(* Logix 5000 project; controller Amvex_Thorpe_Flowmeter vendor 1 type 14 code 106 rev 33.13; software revision 33.01; part 7 of 16 *)

ADD_ON_INSTRUCTION SetCheckpoint   (* revision 0.1, vendor Mecademic Inc., ExecuteEnableInFalse *)
// Inserts a "set checkpoint" command between two moves, so robot status reports that checkpoint id when reaching that command in the queue
VAR_IN_OUT
   RobotInputs : _061D:Meca500_86BDA20B:I:0; {required}
   RobotOutputs : _061D:Meca500_01F88326:O:0; {required}
END_VAR
VAR_INPUT
   Parameter_Value : REAL; {required}
   ExternalStateControl : BOOL; {required}
   ExternalMoveID : INT; {required}
END_VAR
VAR_OUTPUT
   Enabled : BOOL; {visible}
   Sent : BOOL; {visible}
   Buffered : BOOL; {visible}
   Error : BOOL; {visible}
END_VAR
VAR
   InternalMoveID : INT; {access None}
   MoveIDTrig : BOOL; {access None}
   MoveIDUpdated : BOOL; {access None}
   OneShot : DINT; {access None}
   FirstScan : BOOL; {access None}
END_VAR

ROUTINE EnableInFalse   (* ladder *)
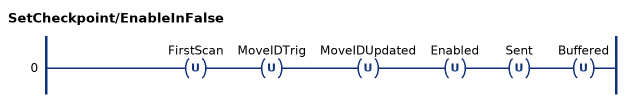
   0: OTU(FirstScan)OTU(MoveIDTrig)OTU(MoveIDUpdated)OTU(Enabled)OTU(Sent)OTU(Buffered);
END_ROUTINE

ROUTINE Logic   (* ladder *)
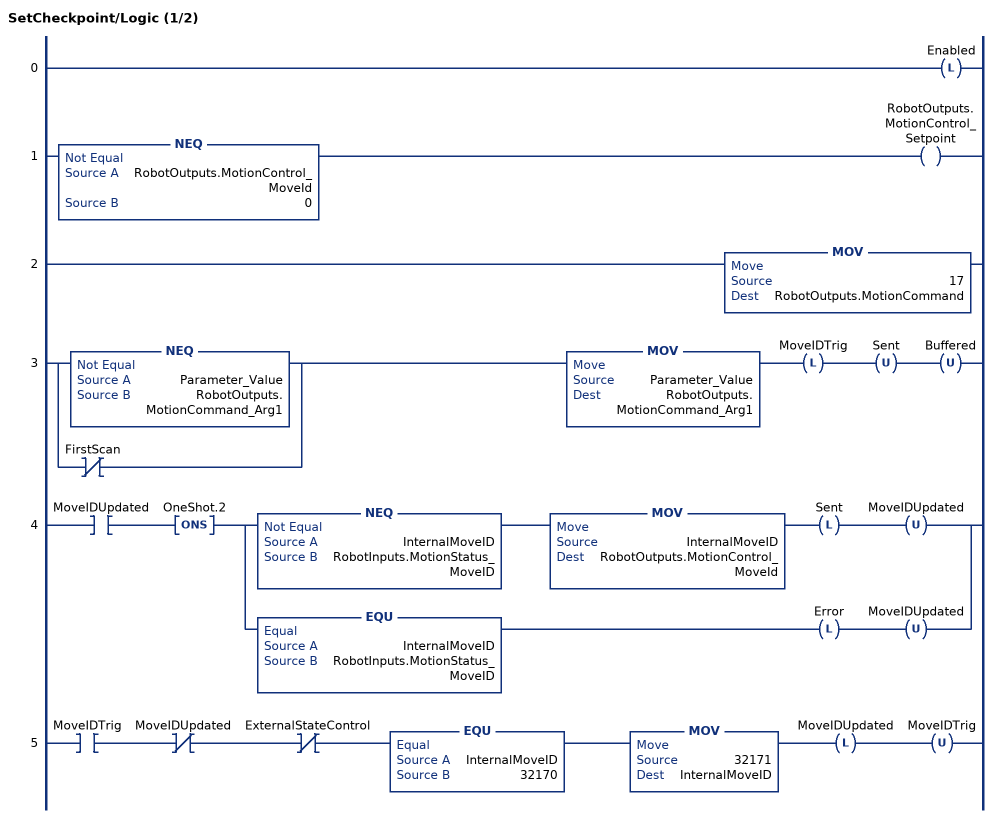
   0: OTL(Enabled);
   1: NEQ(RobotOutputs.MotionControl_MoveId,0)OTE(RobotOutputs.MotionControl_Setpoint);
   2: MOV(17,RobotOutputs.MotionCommand);
   3: [NEQ(Parameter_Value,RobotOutputs.MotionCommand_Arg1) ,XIO(FirstScan) ]MOV(Parameter_Value,RobotOutputs.MotionCommand_Arg1)OTL(MoveIDTrig)OTU(Sent)OTU(Buffered);
   4: XIC(MoveIDUpdated)ONS(OneShot.2)[NEQ(InternalMoveID,RobotInputs.MotionStatus_MoveID) MOV(InternalMoveID,RobotOutputs.MotionControl_MoveId) OTL(Sent) OTU(MoveIDUpdated) ,EQU(InternalMoveID,RobotInputs.MotionStatus_MoveID) OTL(Error) OTU(MoveIDUpdated) ];
   5: XIC(MoveIDTrig)XIO(MoveIDUpdated)XIO(ExternalStateControl)EQU(InternalMoveID,32170)MOV(32171,InternalMoveID)OTL(MoveIDUpdated)OTU(MoveIDTrig);
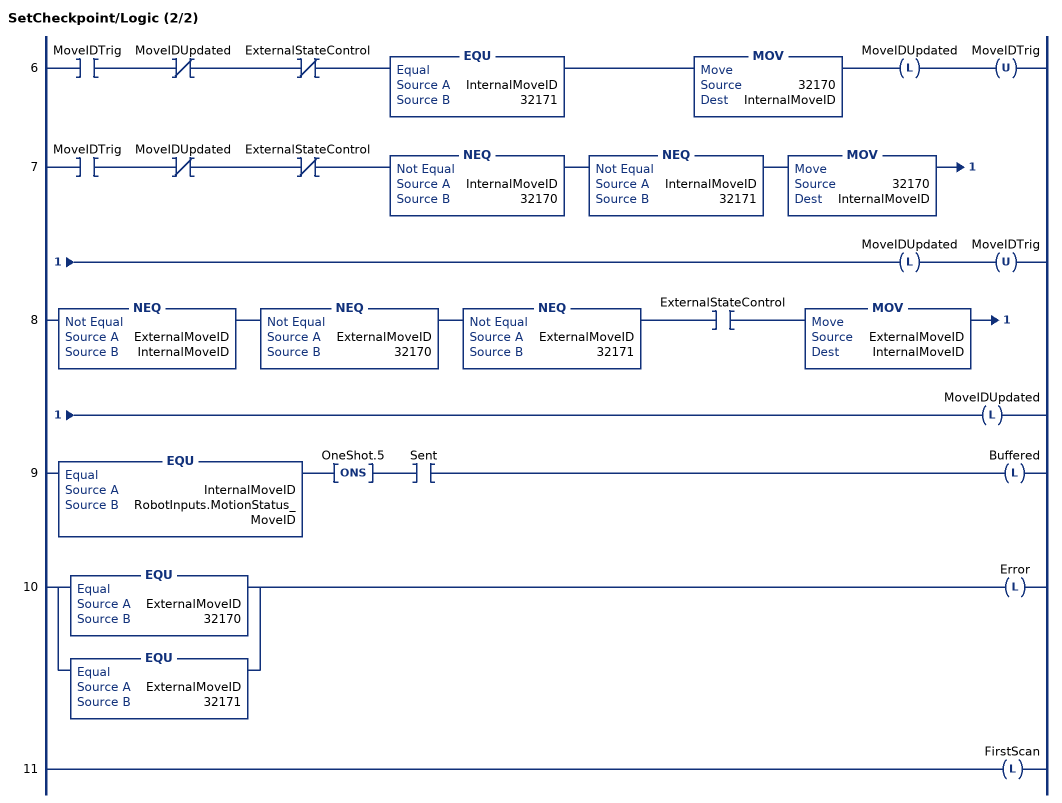
   6: XIC(MoveIDTrig)XIO(MoveIDUpdated)XIO(ExternalStateControl)EQU(InternalMoveID,32171)MOV(32170,InternalMoveID)OTL(MoveIDUpdated)OTU(MoveIDTrig);
   7: XIC(MoveIDTrig)XIO(MoveIDUpdated)XIO(ExternalStateControl)NEQ(InternalMoveID,32170)NEQ(InternalMoveID,32171)MOV(32170,InternalMoveID)OTL(MoveIDUpdated)OTU(MoveIDTrig);
   8: NEQ(ExternalMoveID,InternalMoveID)NEQ(ExternalMoveID,32170)NEQ(ExternalMoveID,32171)XIC(ExternalStateControl)MOV(ExternalMoveID,InternalMoveID)OTL(MoveIDUpdated);
   9: EQU(InternalMoveID,RobotInputs.MotionStatus_MoveID)ONS(OneShot.5)XIC(Sent)OTL(Buffered);
   10: [EQU(ExternalMoveID,32170) ,EQU(ExternalMoveID,32171) ]OTL(Error);
   11: OTL(FirstScan);
END_ROUTINE
END_ADD_ON_INSTRUCTION

ADD_ON_INSTRUCTION SetConf   (* revision 0.1, vendor Mecademic Inc., ExecuteEnableInFalse *)
// Set the desired inverse kinematic config for MovePose. 3 arguments (c1, c3, c5) can be either -1 or 1.
VAR_IN_OUT
   RobotInputs : _061D:Meca500_86BDA20B:I:0; {required}
   RobotOutputs : _061D:Meca500_01F88326:O:0; {required}
END_VAR
VAR_INPUT
   Conf_1 : REAL; {required}
   Conf_2 : REAL; {required}
   Conf_3 : REAL; {required}
   ExternalStateControl : BOOL; {required}
   ExternalMoveID : INT; {required}
END_VAR
VAR_OUTPUT
   Enabled : BOOL; {visible}
   Sent : BOOL; {visible}
   Buffered : BOOL; {visible}
   Error : BOOL; {visible}
END_VAR
VAR
   InternalMoveID : INT; {access None}
   MoveIDTrig : BOOL; {access None}
   MoveIDUpdated : BOOL; {access None}
   OneShot : DINT; {access None}
   FirstScan : BOOL; {access None}
END_VAR

ROUTINE EnableInFalse   (* ladder *)
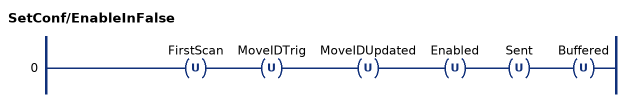
   0: OTU(FirstScan)OTU(MoveIDTrig)OTU(MoveIDUpdated)OTU(Enabled)OTU(Sent)OTU(Buffered);
END_ROUTINE

ROUTINE Logic   (* ladder *)
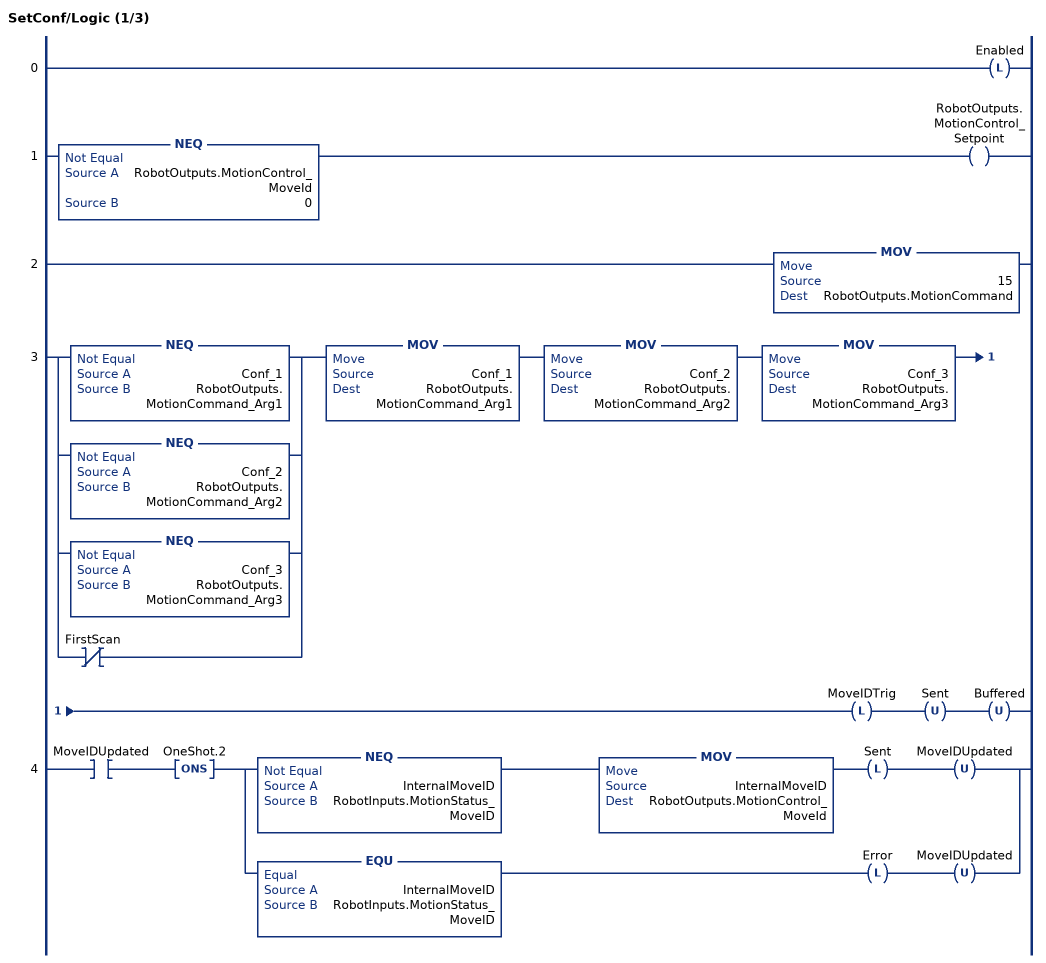
   0: OTL(Enabled);
   1: NEQ(RobotOutputs.MotionControl_MoveId,0)OTE(RobotOutputs.MotionControl_Setpoint);
   2: MOV(15,RobotOutputs.MotionCommand);
   3: [NEQ(Conf_1,RobotOutputs.MotionCommand_Arg1) ,NEQ(Conf_2,RobotOutputs.MotionCommand_Arg2) ,NEQ(Conf_3,RobotOutputs.MotionCommand_Arg3) ,XIO(FirstScan) ]MOV(Conf_1,RobotOutputs.MotionCommand_Arg1)MOV(Conf_2,RobotOutputs.MotionCommand_Arg2)MOV(Conf_3,RobotOutputs.MotionCommand_Arg3)OTL(MoveIDTrig)OTU(Sent)OTU(Buffered);
   4: XIC(MoveIDUpdated)ONS(OneShot.2)[NEQ(InternalMoveID,RobotInputs.MotionStatus_MoveID) MOV(InternalMoveID,RobotOutputs.MotionControl_MoveId) OTL(Sent) OTU(MoveIDUpdated) ,EQU(InternalMoveID,RobotInputs.MotionStatus_MoveID) OTL(Error) OTU(MoveIDUpdated) ];
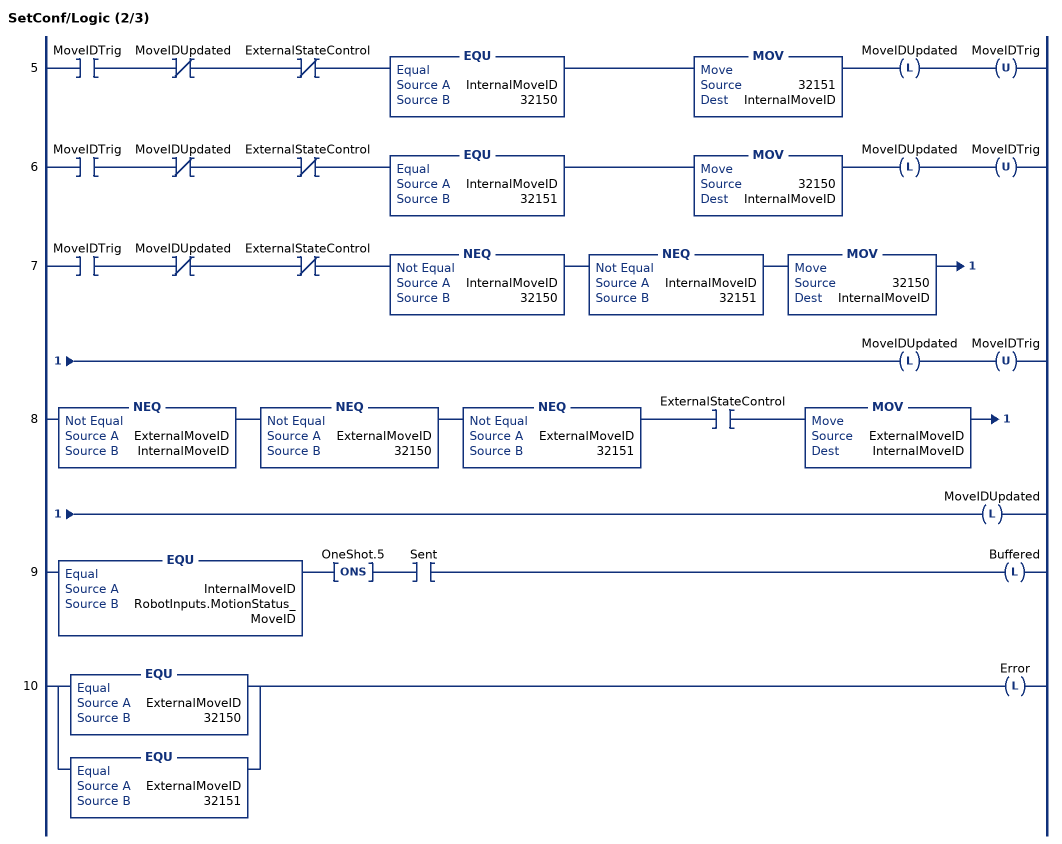
   5: XIC(MoveIDTrig)XIO(MoveIDUpdated)XIO(ExternalStateControl)EQU(InternalMoveID,32150)MOV(32151,InternalMoveID)OTL(MoveIDUpdated)OTU(MoveIDTrig);
   6: XIC(MoveIDTrig)XIO(MoveIDUpdated)XIO(ExternalStateControl)EQU(InternalMoveID,32151)MOV(32150,InternalMoveID)OTL(MoveIDUpdated)OTU(MoveIDTrig);
   7: XIC(MoveIDTrig)XIO(MoveIDUpdated)XIO(ExternalStateControl)NEQ(InternalMoveID,32150)NEQ(InternalMoveID,32151)MOV(32150,InternalMoveID)OTL(MoveIDUpdated)OTU(MoveIDTrig);
   8: NEQ(ExternalMoveID,InternalMoveID)NEQ(ExternalMoveID,32150)NEQ(ExternalMoveID,32151)XIC(ExternalStateControl)MOV(ExternalMoveID,InternalMoveID)OTL(MoveIDUpdated);
   9: EQU(InternalMoveID,RobotInputs.MotionStatus_MoveID)ONS(OneShot.5)XIC(Sent)OTL(Buffered);
   10: [EQU(ExternalMoveID,32150) ,EQU(ExternalMoveID,32151) ]OTL(Error);
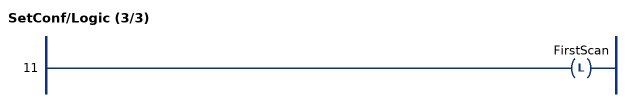
   11: OTL(FirstScan);
END_ROUTINE
END_ADD_ON_INSTRUCTION

ADD_ON_INSTRUCTION SetConfTurn   (* revision 0.1, vendor Mecademic Inc., ExecuteEnableInFalse *)
// Set the last joint desired turn (i.e. which turn should be used during Cartesian moves). Turn 0 uses range ]-180,180].
VAR_IN_OUT
   RobotInputs : _061D:Meca500_86BDA20B:I:0; {required}
   RobotOutputs : _061D:Meca500_01F88326:O:0; {required}
END_VAR
VAR_INPUT
   TurnConf : REAL; {required}
   ExternalStateControl : BOOL; {required}
   ExternalMoveID : INT; {required}
END_VAR
VAR_OUTPUT
   Enabled : BOOL; {visible}
   Sent : BOOL; {visible}
   Buffered : BOOL; {visible}
   Error : BOOL; {visible}
END_VAR
VAR
   InternalMoveID : INT; {access None}
   MoveIDTrig : BOOL; {access None}
   MoveIDUpdated : BOOL; {access None}
   OneShot : DINT; {access None}
   FirstScan : BOOL; {access None}
END_VAR

ROUTINE EnableInFalse   (* ladder *)
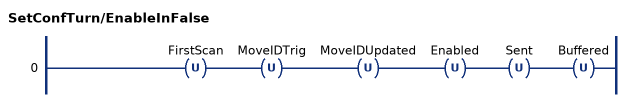
   0: OTU(FirstScan)OTU(MoveIDTrig)OTU(MoveIDUpdated)OTU(Enabled)OTU(Sent)OTU(Buffered);
END_ROUTINE

ROUTINE Logic   (* ladder *)
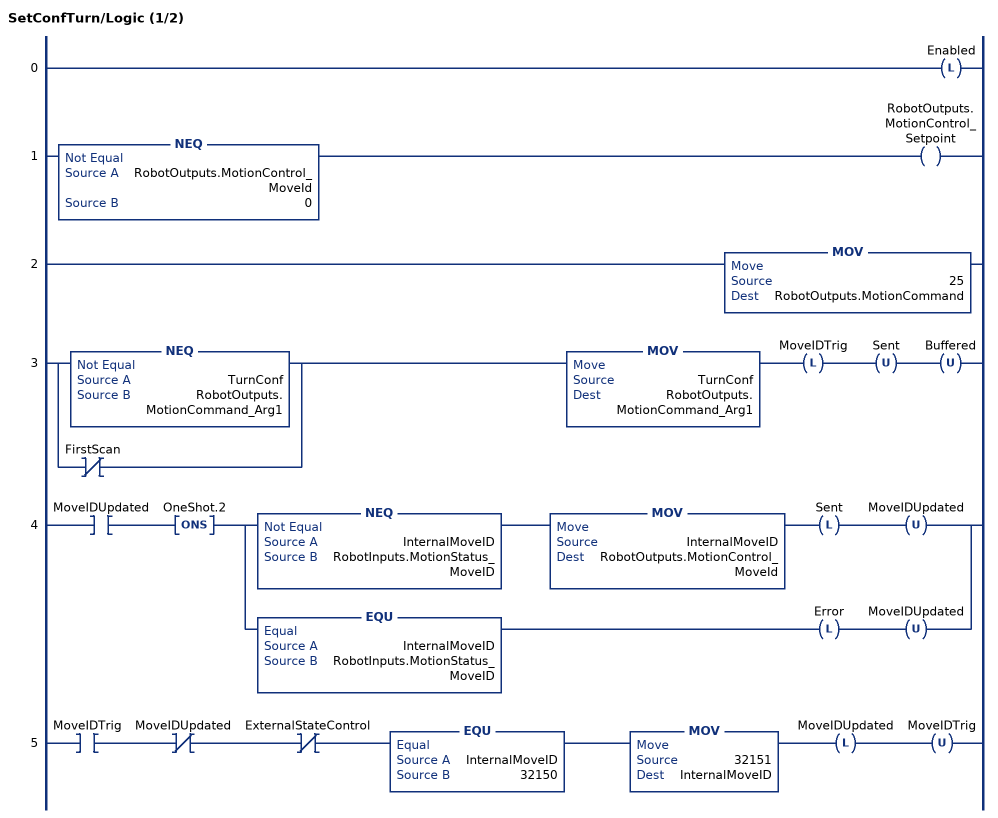
   0: OTL(Enabled);
   1: NEQ(RobotOutputs.MotionControl_MoveId,0)OTE(RobotOutputs.MotionControl_Setpoint);
   2: MOV(25,RobotOutputs.MotionCommand);
   3: [NEQ(TurnConf,RobotOutputs.MotionCommand_Arg1) ,XIO(FirstScan) ]MOV(TurnConf,RobotOutputs.MotionCommand_Arg1)OTL(MoveIDTrig)OTU(Sent)OTU(Buffered);
   4: XIC(MoveIDUpdated)ONS(OneShot.2)[NEQ(InternalMoveID,RobotInputs.MotionStatus_MoveID) MOV(InternalMoveID,RobotOutputs.MotionControl_MoveId) OTL(Sent) OTU(MoveIDUpdated) ,EQU(InternalMoveID,RobotInputs.MotionStatus_MoveID) OTL(Error) OTU(MoveIDUpdated) ];
   5: XIC(MoveIDTrig)XIO(MoveIDUpdated)XIO(ExternalStateControl)EQU(InternalMoveID,32150)MOV(32151,InternalMoveID)OTL(MoveIDUpdated)OTU(MoveIDTrig);
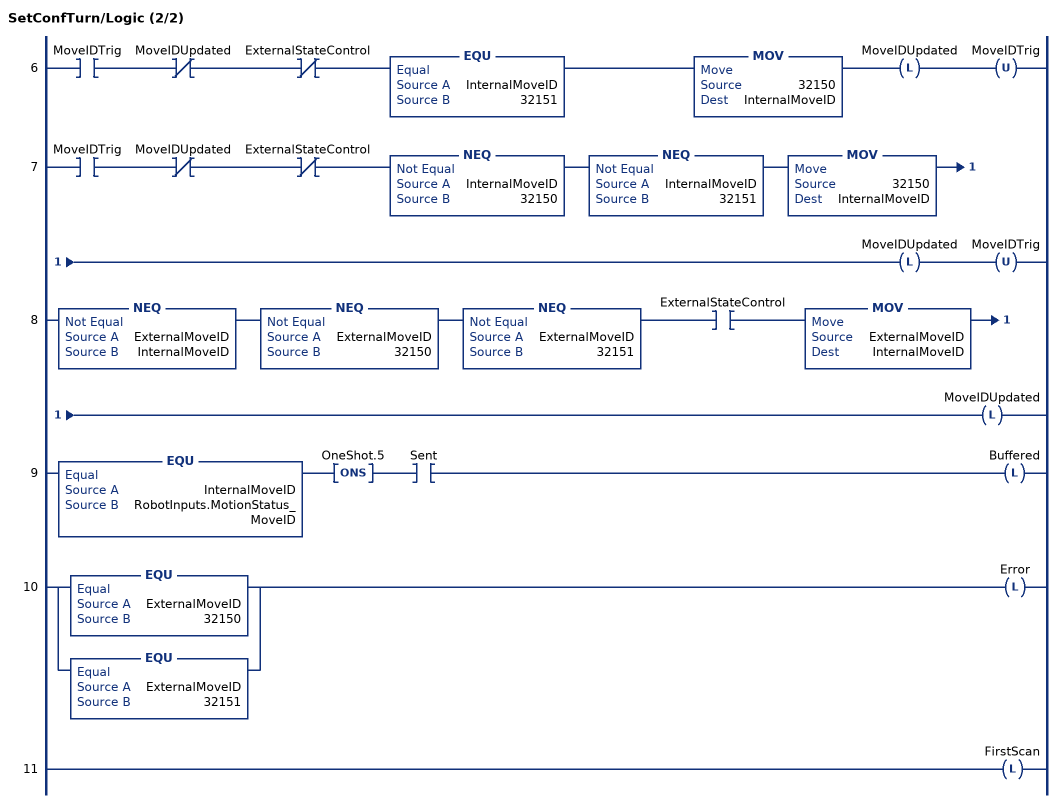
   6: XIC(MoveIDTrig)XIO(MoveIDUpdated)XIO(ExternalStateControl)EQU(InternalMoveID,32151)MOV(32150,InternalMoveID)OTL(MoveIDUpdated)OTU(MoveIDTrig);
   7: XIC(MoveIDTrig)XIO(MoveIDUpdated)XIO(ExternalStateControl)NEQ(InternalMoveID,32150)NEQ(InternalMoveID,32151)MOV(32150,InternalMoveID)OTL(MoveIDUpdated)OTU(MoveIDTrig);
   8: NEQ(ExternalMoveID,InternalMoveID)NEQ(ExternalMoveID,32150)NEQ(ExternalMoveID,32151)XIC(ExternalStateControl)MOV(ExternalMoveID,InternalMoveID)OTL(MoveIDUpdated);
   9: EQU(InternalMoveID,RobotInputs.MotionStatus_MoveID)ONS(OneShot.5)XIC(Sent)OTL(Buffered);
   10: [EQU(ExternalMoveID,32150) ,EQU(ExternalMoveID,32151) ]OTL(Error);
   11: OTL(FirstScan);
END_ROUTINE
END_ADD_ON_INSTRUCTION

ADD_ON_INSTRUCTION SetGripperForce   (* revision 0.1, vendor Mecademic Inc., ExecuteEnableInFalse *)
// Limit the grip force of the gripper in percent
VAR_IN_OUT
   RobotInputs : _061D:Meca500_86BDA20B:I:0; {required}
   RobotOutputs : _061D:Meca500_01F88326:O:0; {required}
END_VAR
VAR_INPUT
   Parameter_Value : REAL; {required}
   ExternalStateControl : BOOL; {required}
   ExternalMoveID : INT; {required}
END_VAR
VAR_OUTPUT
   Enabled : BOOL; {visible}
   Sent : BOOL; {visible}
   Buffered : BOOL; {visible}
   Error : BOOL; {visible}
END_VAR
VAR
   InternalMoveID : INT; {access None}
   MoveIDTrig : BOOL; {access None}
   MoveIDUpdated : BOOL; {access None}
   OneShot : DINT; {access None}
   FirstScan : BOOL; {access None}
END_VAR

ROUTINE EnableInFalse   (* ladder *)
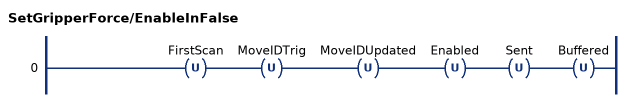
   0: OTU(FirstScan)OTU(MoveIDTrig)OTU(MoveIDUpdated)OTU(Enabled)OTU(Sent)OTU(Buffered);
END_ROUTINE

ROUTINE Logic   (* ladder *)
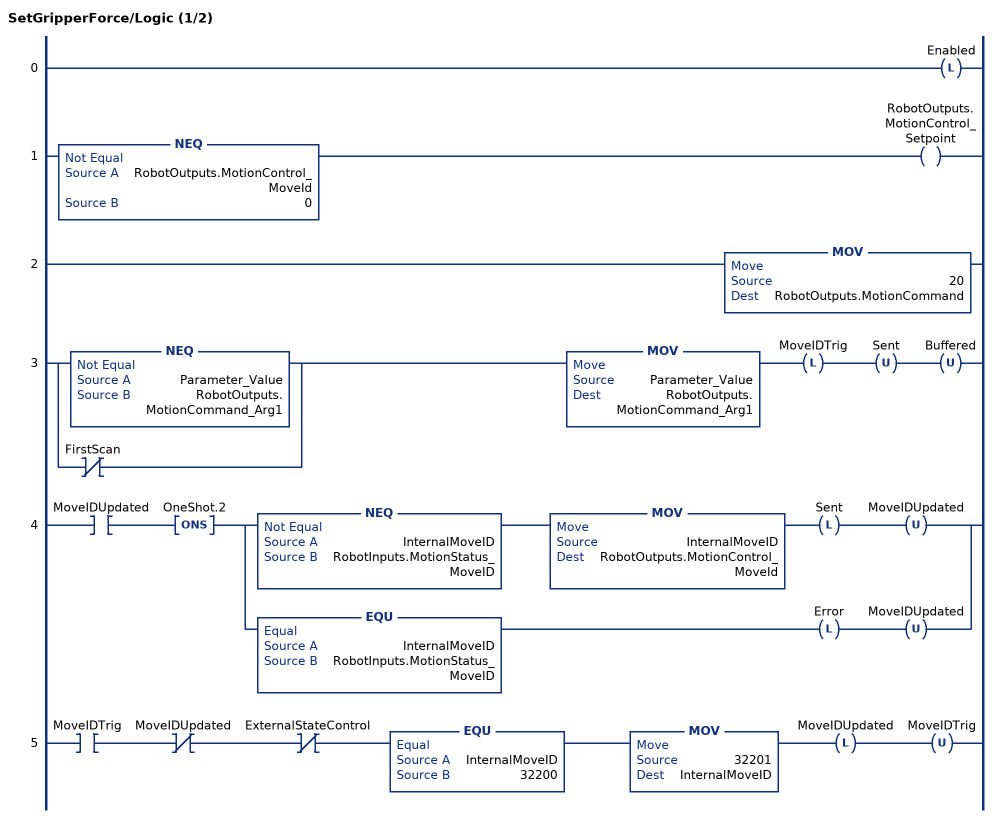
   0: OTL(Enabled);
   1: NEQ(RobotOutputs.MotionControl_MoveId,0)OTE(RobotOutputs.MotionControl_Setpoint);
   2: MOV(20,RobotOutputs.MotionCommand);
   3: [NEQ(Parameter_Value,RobotOutputs.MotionCommand_Arg1) ,XIO(FirstScan) ]MOV(Parameter_Value,RobotOutputs.MotionCommand_Arg1)OTL(MoveIDTrig)OTU(Sent)OTU(Buffered);
   4: XIC(MoveIDUpdated)ONS(OneShot.2)[NEQ(InternalMoveID,RobotInputs.MotionStatus_MoveID) MOV(InternalMoveID,RobotOutputs.MotionControl_MoveId) OTL(Sent) OTU(MoveIDUpdated) ,EQU(InternalMoveID,RobotInputs.MotionStatus_MoveID) OTL(Error) OTU(MoveIDUpdated) ];
   5: XIC(MoveIDTrig)XIO(MoveIDUpdated)XIO(ExternalStateControl)EQU(InternalMoveID,32200)MOV(32201,InternalMoveID)OTL(MoveIDUpdated)OTU(MoveIDTrig);
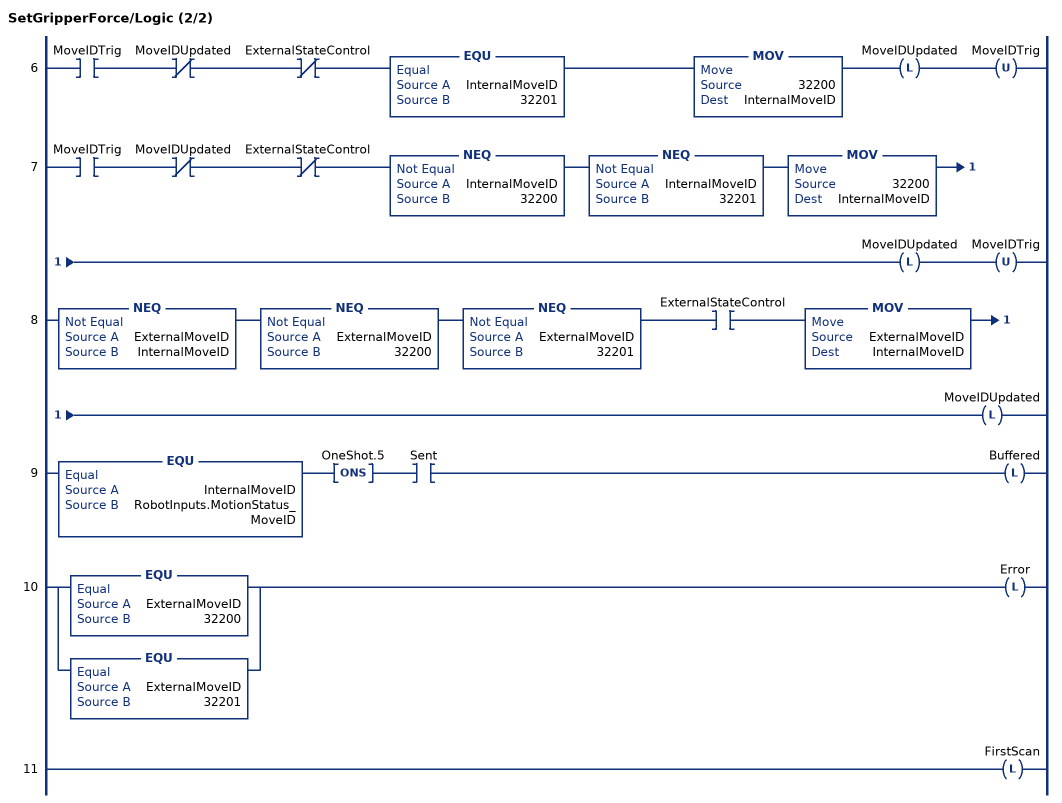
   6: XIC(MoveIDTrig)XIO(MoveIDUpdated)XIO(ExternalStateControl)EQU(InternalMoveID,32201)MOV(32200,InternalMoveID)OTL(MoveIDUpdated)OTU(MoveIDTrig);
   7: XIC(MoveIDTrig)XIO(MoveIDUpdated)XIO(ExternalStateControl)NEQ(InternalMoveID,32200)NEQ(InternalMoveID,32201)MOV(32200,InternalMoveID)OTL(MoveIDUpdated)OTU(MoveIDTrig);
   8: NEQ(ExternalMoveID,InternalMoveID)NEQ(ExternalMoveID,32200)NEQ(ExternalMoveID,32201)XIC(ExternalStateControl)MOV(ExternalMoveID,InternalMoveID)OTL(MoveIDUpdated);
   9: EQU(InternalMoveID,RobotInputs.MotionStatus_MoveID)ONS(OneShot.5)XIC(Sent)OTL(Buffered);
   10: [EQU(ExternalMoveID,32200) ,EQU(ExternalMoveID,32201) ]OTL(Error);
   11: OTL(FirstScan);
END_ROUTINE
END_ADD_ON_INSTRUCTION

ADD_ON_INSTRUCTION SetGripperVel   (* revision 0.1, vendor Mecademic Inc., ExecuteEnableInFalse *)
// Limit the velocity of the gripper fingers in percent
VAR_IN_OUT
   RobotInputs : _061D:Meca500_86BDA20B:I:0; {required}
   RobotOutputs : _061D:Meca500_01F88326:O:0; {required}
END_VAR
VAR_INPUT
   Parameter_Value : REAL; {required}
   ExternalStateControl : BOOL; {required}
   ExternalMoveID : INT; {required}
END_VAR
VAR_OUTPUT
   Enabled : BOOL; {visible}
   Sent : BOOL; {visible}
   Buffered : BOOL; {visible}
   Error : BOOL; {visible}
END_VAR
VAR
   InternalMoveID : INT; {access None}
   MoveIDTrig : BOOL; {access None}
   MoveIDUpdated : BOOL; {access None}
   OneShot : DINT; {access None}
   FirstScan : BOOL; {access None}
END_VAR

ROUTINE EnableInFalse   (* ladder *)
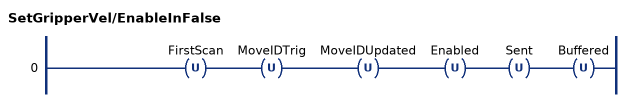
   0: OTU(FirstScan)OTU(MoveIDTrig)OTU(MoveIDUpdated)OTU(Enabled)OTU(Sent)OTU(Buffered);
END_ROUTINE

ROUTINE Logic   (* ladder *)
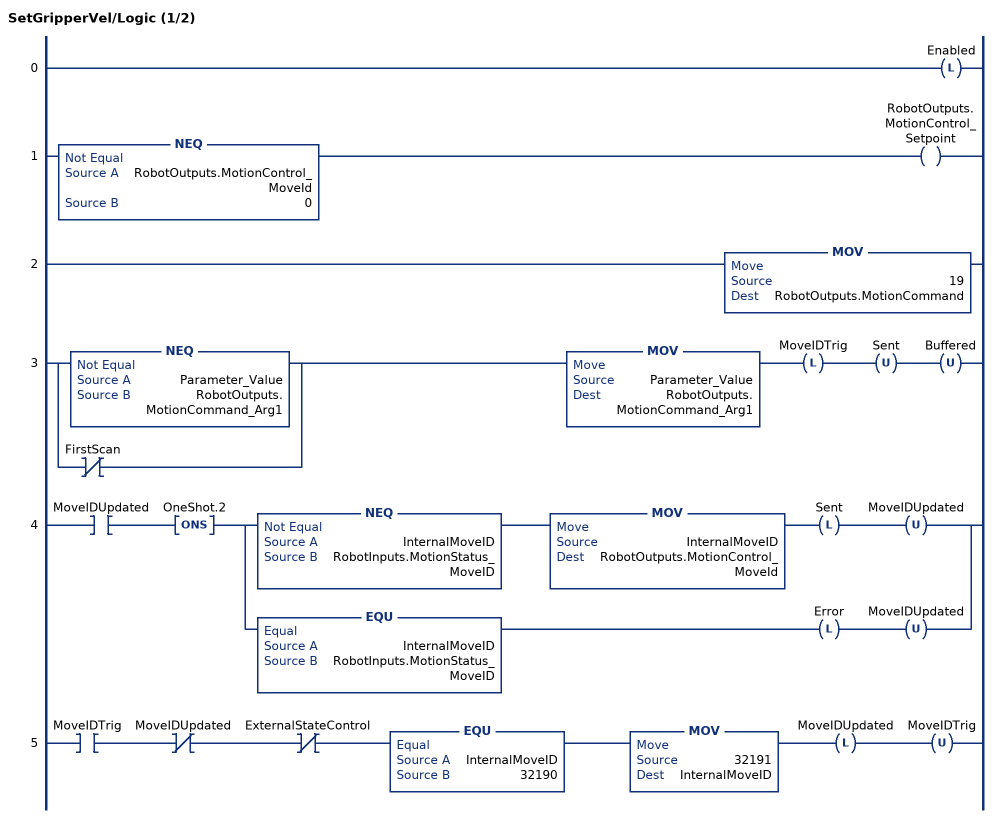
   0: OTL(Enabled);
   1: NEQ(RobotOutputs.MotionControl_MoveId,0)OTE(RobotOutputs.MotionControl_Setpoint);
   2: MOV(19,RobotOutputs.MotionCommand);
   3: [NEQ(Parameter_Value,RobotOutputs.MotionCommand_Arg1) ,XIO(FirstScan) ]MOV(Parameter_Value,RobotOutputs.MotionCommand_Arg1)OTL(MoveIDTrig)OTU(Sent)OTU(Buffered);
   4: XIC(MoveIDUpdated)ONS(OneShot.2)[NEQ(InternalMoveID,RobotInputs.MotionStatus_MoveID) MOV(InternalMoveID,RobotOutputs.MotionControl_MoveId) OTL(Sent) OTU(MoveIDUpdated) ,EQU(InternalMoveID,RobotInputs.MotionStatus_MoveID) OTL(Error) OTU(MoveIDUpdated) ];
   5: XIC(MoveIDTrig)XIO(MoveIDUpdated)XIO(ExternalStateControl)EQU(InternalMoveID,32190)MOV(32191,InternalMoveID)OTL(MoveIDUpdated)OTU(MoveIDTrig);
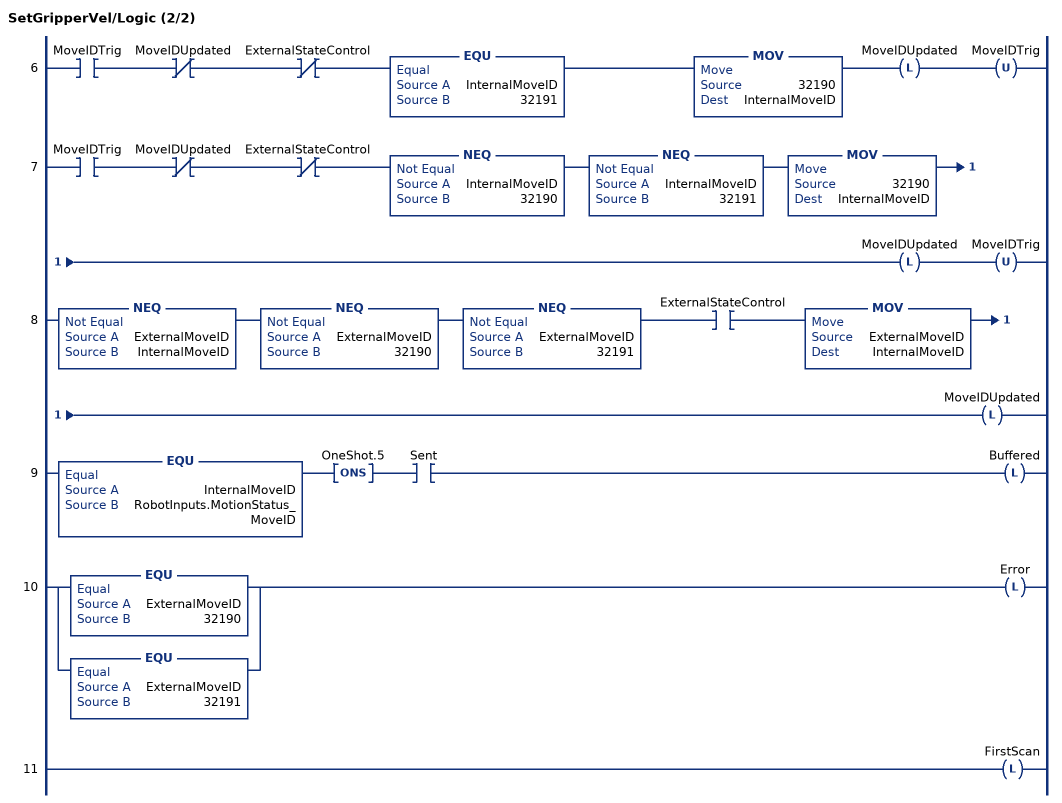
   6: XIC(MoveIDTrig)XIO(MoveIDUpdated)XIO(ExternalStateControl)EQU(InternalMoveID,32191)MOV(32190,InternalMoveID)OTL(MoveIDUpdated)OTU(MoveIDTrig);
   7: XIC(MoveIDTrig)XIO(MoveIDUpdated)XIO(ExternalStateControl)NEQ(InternalMoveID,32190)NEQ(InternalMoveID,32191)MOV(32190,InternalMoveID)OTL(MoveIDUpdated)OTU(MoveIDTrig);
   8: NEQ(ExternalMoveID,InternalMoveID)NEQ(ExternalMoveID,32190)NEQ(ExternalMoveID,32191)XIC(ExternalStateControl)MOV(ExternalMoveID,InternalMoveID)OTL(MoveIDUpdated);
   9: EQU(InternalMoveID,RobotInputs.MotionStatus_MoveID)ONS(OneShot.5)XIC(Sent)OTL(Buffered);
   10: [EQU(ExternalMoveID,32190) ,EQU(ExternalMoveID,32191) ]OTL(Error);
   11: OTL(FirstScan);
END_ROUTINE
END_ADD_ON_INSTRUCTION

ADD_ON_INSTRUCTION SetJointAcc   (* revision 0.1, vendor Mecademic Inc., ExecuteEnableInFalse *)
// Set joint acceleration in percent (for MovePost and MoveJoint only)
VAR_IN_OUT
   RobotInputs : _061D:Meca500_86BDA20B:I:0; {required}
   RobotOutputs : _061D:Meca500_01F88326:O:0; {required}
END_VAR
VAR_INPUT
   Parameter_Value : REAL; {required}
   ExternalStateControl : BOOL; {required}
   ExternalMoveID : INT; {required}
END_VAR
VAR_OUTPUT
   Enabled : BOOL; {visible}
   Sent : BOOL; {visible}
   Buffered : BOOL; {visible}
   Error : BOOL; {visible}
END_VAR
VAR
   InternalMoveID : INT; {access None}
   MoveIDTrig : BOOL; {access None}
   MoveIDUpdated : BOOL; {access None}
   OneShot : DINT; {access None}
   FirstScan : BOOL; {access None}
END_VAR

ROUTINE EnableInFalse   (* ladder *)
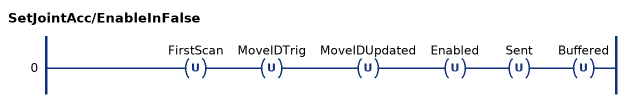
   0: OTU(FirstScan)OTU(MoveIDTrig)OTU(MoveIDUpdated)OTU(Enabled)OTU(Sent)OTU(Buffered);
END_ROUTINE

ROUTINE Logic   (* ladder *)
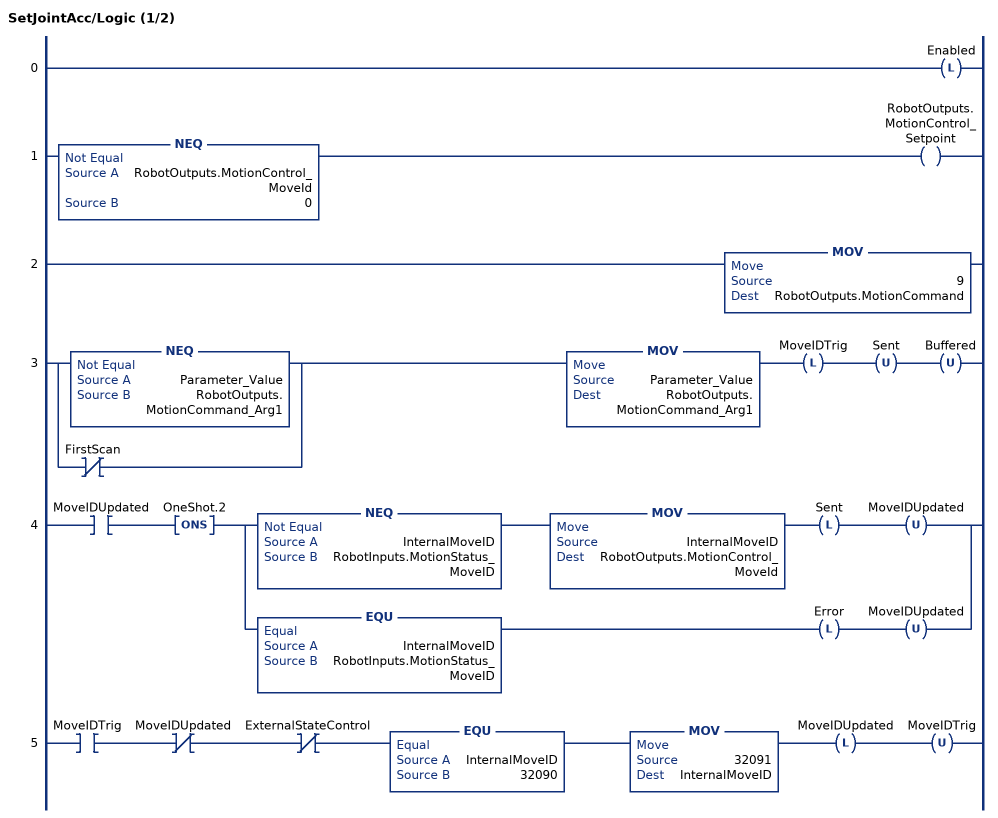
   0: OTL(Enabled);
   1: NEQ(RobotOutputs.MotionControl_MoveId,0)OTE(RobotOutputs.MotionControl_Setpoint);
   2: MOV(9,RobotOutputs.MotionCommand);
   3: [NEQ(Parameter_Value,RobotOutputs.MotionCommand_Arg1) ,XIO(FirstScan) ]MOV(Parameter_Value,RobotOutputs.MotionCommand_Arg1)OTL(MoveIDTrig)OTU(Sent)OTU(Buffered);
   4: XIC(MoveIDUpdated)ONS(OneShot.2)[NEQ(InternalMoveID,RobotInputs.MotionStatus_MoveID) MOV(InternalMoveID,RobotOutputs.MotionControl_MoveId) OTL(Sent) OTU(MoveIDUpdated) ,EQU(InternalMoveID,RobotInputs.MotionStatus_MoveID) OTL(Error) OTU(MoveIDUpdated) ];
   5: XIC(MoveIDTrig)XIO(MoveIDUpdated)XIO(ExternalStateControl)EQU(InternalMoveID,32090)MOV(32091,InternalMoveID)OTL(MoveIDUpdated)OTU(MoveIDTrig);
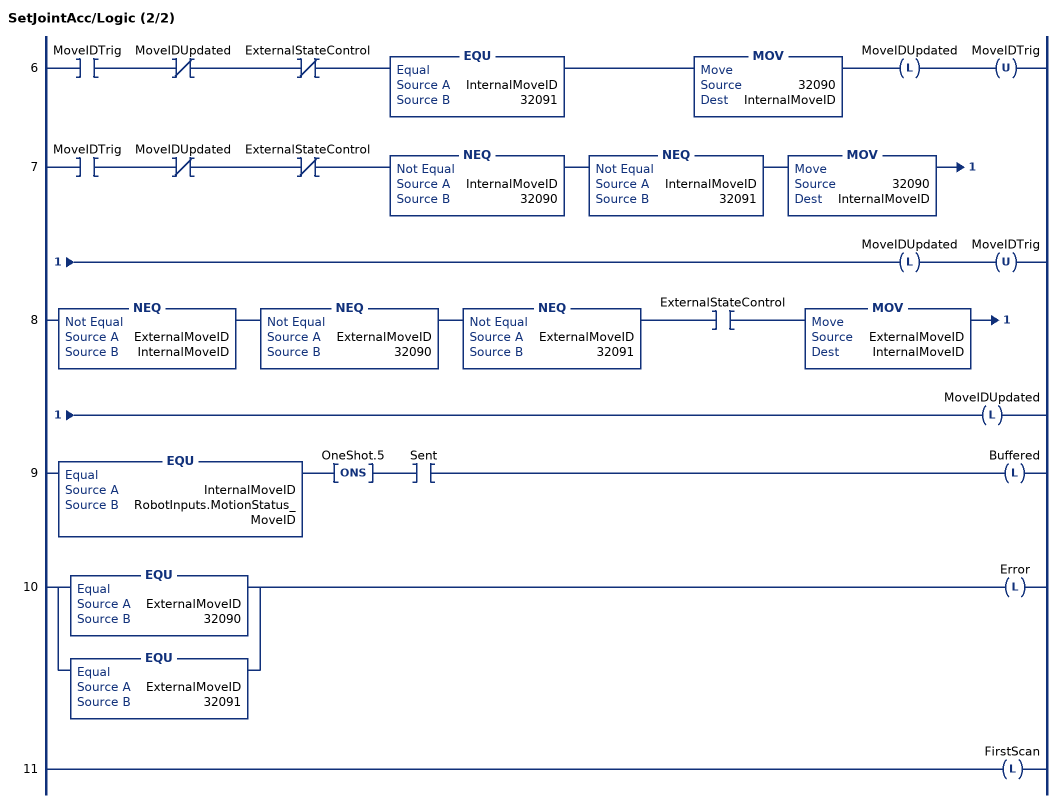
   6: XIC(MoveIDTrig)XIO(MoveIDUpdated)XIO(ExternalStateControl)EQU(InternalMoveID,32091)MOV(32090,InternalMoveID)OTL(MoveIDUpdated)OTU(MoveIDTrig);
   7: XIC(MoveIDTrig)XIO(MoveIDUpdated)XIO(ExternalStateControl)NEQ(InternalMoveID,32090)NEQ(InternalMoveID,32091)MOV(32090,InternalMoveID)OTL(MoveIDUpdated)OTU(MoveIDTrig);
   8: NEQ(ExternalMoveID,InternalMoveID)NEQ(ExternalMoveID,32090)NEQ(ExternalMoveID,32091)XIC(ExternalStateControl)MOV(ExternalMoveID,InternalMoveID)OTL(MoveIDUpdated);
   9: EQU(InternalMoveID,RobotInputs.MotionStatus_MoveID)ONS(OneShot.5)XIC(Sent)OTL(Buffered);
   10: [EQU(ExternalMoveID,32090) ,EQU(ExternalMoveID,32091) ]OTL(Error);
   11: OTL(FirstScan);
END_ROUTINE
END_ADD_ON_INSTRUCTION
